// TIA Portal V20 export
DATA_BLOCK "DB_HMISetting"   // DB1306
{ S7_Optimized_Access := 'FALSE' }
AUTHOR : DAT
NAME : IHM_SETT
// stored: AutoNumber false
   VAR RETAIN
      GasAssistSetPoint : Real;
      CoolingVentilatorSetpoint : Real;   // @Precision:0 @Unit:% @Min:0 @Max:100
      TemperatureCoolingSetpoint : Real;   // @Precision:1 @Unit:°C @Min:0 @Max:50
      BlowingSetpoint : Real;   // @Precision:0 @Unit:ms @Min:0 @Max:500
      WorkingMode : Struct
         EmptyingReq : Bool;
      END_STRUCT;
      Sonplas : Struct
         LimitMax : Real;
         LimitCtrlMax : Real;
         LimitCtrlMin : Real;
         LimitMin : Real;
         CorrectionMax : Real;
         CorrectionMin : Real;
      END_STRUCT;
      LockDoorReq : Bool;
      UnlockDoorReq : Bool;
      StartAutoReq : Bool;
      StopAutoReq : Bool;
      Shuttle1Enable : Bool;
      Shuttle2Enable : Bool;
   END_VAR
BEGIN
END_DATA_BLOCK
